		160: //Vision capture tray fiducial 1
			arrStepStatus[7] := 'Step 7: Trigger Vision Capture';
			tonStepTimer(IN:=TRUE, PT:=T#999999S);
			IF NOT G_MachineControl.stMachineOperateMode.DRYRUN THEN
				G_Vision.V20_bRespone := FALSE;
				G_Vision.V20_sSendCmd := 'TRG,2';  
				G_Vision.V20_bTrigger := TRUE;	
			END_IF			
			iStep := 170;
		
		170: //Waiting vision capture done
			tonTimeOut(IN:= TRUE,PT:= tTimeOut);
			IF G_Vision.V20_bRespone OR G_MachineControl.stMachineOperateMode.DRYRUN THEN
				tonTimeOut(IN:= FALSE);
				G_Vision.V20_bTrigger := FALSE;
				arrStepUsedTime[7] := tonStepTimer.ET;
				tonStepTimer(IN:=FALSE);
				iStep := 180;
			ELSIF tonTimeOut.Q THEN
				tonTimeOut(IN:= FALSE);
				G_Vision.V20_bTrigger := FALSE;	
				G_Error.E20_VisionTimeOutInspection	:= TRUE;
				iStep := 160;
			END_IF
			
		180:
			G_Robot.RobotKukaCmd.rRobotPlace_X := G_Values.VA20_stTrayPosition.stFiducialDistance2Value.Xpos;
			G_Robot.RobotKukaCmd.rRobotPlace_Y := G_Values.VA20_stTrayPosition.stFiducialDistance2Value.Ypos;
			G_Robot.RobotKukaCmd.rRobotPlace_Z := 0; //G_Values.VA20_stTrayPosition.stFiducialDistance2Value.Zpos;
			G_Robot.RobotKukaCmd.rRobotPlace_A := G_Values.VA20_stTrayPosition.stFiducialDistance2Value.Apos;
			iStep := 190;
			
		190: //Robot move to tray fiducial 2
			arrStepStatus[8] := 'Step 8: Robot go to tray fiducial 2';
			tonStepTimer(IN:=TRUE, PT:=T#999999S);
			G_Robot.RobotKukaCmd.bRobotTrayFiducial2 := TRUE;
			iStep := 200; 
			
		200:
			IF NOT G_Robot.RobotKukaCmd.bRobotTrayFiducial2Done THEN
				iStep := 210;
			END_IF
			
		210://Robot move tray fiducial 2 done
			tonTimeOut(IN:= TRUE,PT:= tTimeOut);
			IF G_Robot.RobotKukaCmd.bRobotTrayFiducial2Done THEN
				tonTimeOut(IN:= FALSE);
				G_Robot.RobotKukaCmd.bRobotTrayFiducial2 := FALSE;
				arrStepUsedTime[8] := tonStepTimer.ET;
				tonStepTimer(IN:=FALSE);
				iStep := 220;
			ELSIF tonTimeOut.Q THEN
				tonTimeOut(IN:= FALSE);
				G_Robot.RobotKukaCmd.bRobotTrayFiducial2 := FALSE;
				G_Error.E20_RobotTimeOutFailToTrayFiducial_2 := TRUE;
				iStep := 180;
			END_IF
			
		220: //Vision capture tray fiducial 2
			arrStepStatus[9] := 'Step 9: Trigger Vision Capture';
			tonStepTimer(IN:=TRUE, PT:=T#999999S);
			IF NOT G_MachineControl.stMachineOperateMode.DRYRUN THEN
				G_Vision.V20_bRespone := FALSE;
				G_Vision.V20_sSendCmd := 'TRG,3'; 
				G_Vision.V20_bTrigger := TRUE;	
			END_IF				
			iStep := 230;
		
		230: //Waiting vision capture done
			tonTimeOut(IN:= TRUE,PT:= tTimeOut);
			IF G_Vision.V20_bRespone OR G_MachineControl.stMachineOperateMode.DRYRUN THEN
				tonTimeOut(IN:= FALSE);
				G_Vision.V20_bTrigger := FALSE;
				arrStepUsedTime[9] := tonStepTimer.ET;
				tonStepTimer(IN:=FALSE);
				iStep := 240;
			ELSIF tonTimeOut.Q THEN
				tonTimeOut(IN:= FALSE);
				G_Vision.V20_bTrigger := FALSE;	
				G_Error.E20_VisionTimeOutInspection	:= TRUE;
				iStep := 220;
			END_IF
			
		240:
			IF NOT G_MachineControl.stMachineOperateMode.DRYRUN THEN
				G_Robot.RobotKukaCmd.rRobotPlace_X := G_Vision.V20_stTrayPosition.stPocket.Xpos;
				G_Robot.RobotKukaCmd.rRobotPlace_Y := G_Vision.V20_stTrayPosition.stPocket.Ypos;
				G_Robot.RobotKukaCmd.rRobotPlace_Z := G_Values.VA20_rTrayZaxisPick; //G_Vision.V20_stTrayPosition.stPocket.Zpos;
				G_Robot.RobotKukaCmd.rRobotPlace_A := G_Vision.V20_stTrayPosition.stPocket.Apos;
			ELSIF G_MachineControl.stMachineOperateMode.DRYRUN THEN
				G_Robot.RobotKukaCmd.rRobotPlace_X := G_Values.VA20_stTrayPosition.stPocket.Xpos;
				G_Robot.RobotKukaCmd.rRobotPlace_Y := G_Values.VA20_stTrayPosition.stPocket.Ypos;
				G_Robot.RobotKukaCmd.rRobotPlace_Z := G_Values.VA20_rTrayZaxisPick; //G_Values.VA20_stTrayPosition.stPocket.Zpos;
				G_Robot.RobotKukaCmd.rRobotPlace_A := G_Values.VA20_stTrayPosition.stPocket.Apos;
			END_IF
			iStep := 250;
			
		250: //Robot move to pick PCBA
			arrStepStatus[10] := 'Step 10: Robot go to pick PCBA';
			tonStepTimer(IN:=TRUE, PT:=T#999999S);
			G_Robot.RobotKukaCmd.bRobotPickPCBA := TRUE;
			iStep := 260; 
			
		260:
			IF NOT G_Robot.RobotKukaCmd.bRobotPickPCBADone THEN
				iStep := 270;
			END_IF
			
		270://Robot move pick PCBA
			tonTimeOut(IN:= TRUE,PT:= tTimeOut);
			IF G_Robot.RobotKukaCmd.bRobotPickPCBADone THEN
				tonTimeOut(IN:= FALSE);
				G_Auto.A20_bTrayFinish := TRUE;
				G_Robot.RobotKukaCmd.bRobotPickPCBA := FALSE;
				arrStepUsedTime[10] := tonStepTimer.ET;
				tonStepTimer(IN:=FALSE);
				iStep := 280;
			ELSIF tonTimeOut.Q THEN
				tonTimeOut(IN:= FALSE);
				G_Robot.RobotKukaCmd.bRobotPickPCBA := FALSE;
				G_Error.E20_RObotTimeOutFailToPickPCBA := TRUE;
				iStep := 240;
			END_IF
			
		280:
			IF NOT G_MachineControl.stMachineOperateMode.DRYRUN THEN
				G_Robot.RobotKukaCmd.rRobotPlace_X := G_Vision.V20_stPalletPosition.stPocket.Xpos;
				G_Robot.RobotKukaCmd.rRobotPlace_Y := G_Vision.V20_stPalletPosition.stPocket.Ypos;
				G_Robot.RobotKukaCmd.rRobotPlace_Z := G_Values.VA20_rTrayZaxisPick; //G_Vision.V20_stPalletPosition.stPocket.Zpos;
				G_Robot.RobotKukaCmd.rRobotPlace_A := G_Vision.V20_stPalletPosition.stPocket.Apos;
			ELSIF G_MachineControl.stMachineOperateMode.DRYRUN THEN
				G_Robot.RobotKukaCmd.rRobotPlace_X := G_Values.VA20_stPalletPosition.stPocket.Xpos;
				G_Robot.RobotKukaCmd.rRobotPlace_Y := G_Values.VA20_stPalletPosition.stPocket.Ypos;
				G_Robot.RobotKukaCmd.rRobotPlace_Z := G_Values.VA20_rTrayZaxisPick; //G_Values.VA20_stPalletPosition.stPocket.Zpos;
				G_Robot.RobotKukaCmd.rRobotPlace_A := G_Values.VA20_stPalletPosition.stPocket.Apos;
			END_IF
			iStep := 290;
			
		290: //Robot place pcba
			arrStepStatus[11] := 'Step 11: Robot go to place PCBA';
			tonStepTimer(IN:=TRUE, PT:=T#999999S);
			G_Robot.RobotKukaCmd.bRobotPlacePCBA := TRUE;
			iStep := 300;
			
		300:
			IF NOT G_Robot.RobotKukaCmd.bRobotPlacePCBADone THEN
				iStep := 310;
			END_IF
			
		310: //Robot place pcba done
			tonTimeOut(IN:= TRUE,PT:= tTimeOut);
			IF G_Robot.RobotKukaCmd.bRobotPlacePCBADone THEN
				tonTimeOut(IN:= FALSE);
				G_Robot.RobotKukaCmd.bRobotPlacePCBA := FALSE;
				arrStepUsedTime[11] := tonStepTimer.ET;
				tonStepTimer(IN:=FALSE);
				iStep := 320;
			ELSIF tonTimeOut.Q THEN
				tonTimeOut(IN:= FALSE);
				G_Robot.RobotKukaCmd.bRobotPlacePCBA := FALSE;
				G_Error.E20_RobotTimeOutFailToPlacePCBA := TRUE;
				iStep := 280;
			END_IF
			
		320: //Robot go standby pallet
			arrStepStatus[12] := 'Step 12: Robot go to standby';
			tonStepTimer(IN:=TRUE, PT:=T#999999S);
			G_Robot.RobotKukaCmd.bRobotStandbyAtPallet := TRUE;
			iStep := 330;
			
		330:
			IF NOT G_Robot.RobotKukaCmd.bRobotStandbyAtPalletDone THEN
				iStep := 340;
			END_IF
			
		340: //Robot go standby pallet done
			tonTimeOut(IN:= TRUE,PT:= tTimeOut);
			IF G_Robot.RobotKukaCmd.bRobotStandbyAtPalletDone THEN
				tonTimeOut(IN:= FALSE);
				G_Robot.RobotKukaCmd.bRobotStandbyAtPallet := FALSE;
				arrStepUsedTime[12] := tonStepTimer.ET;
				tonStepTimer(IN:=FALSE);
				iStep := 999;
			ELSIF tonTimeOut.Q THEN
				tonTimeOut(IN:= FALSE);
				G_Robot.RobotKukaCmd.bRobotStandbyAtPallet := FALSE;
				G_Error.E20_RobotTimeOutFailToStandbyPallet := TRUE;
				iStep := 280;
			END_IF		
			
		999://Job Done
			G_MachineControl.arrstStationControl[2].bJobDone := TRUE;
			iStep := 0;	
			
		1000: //Robot go to standby at pallet
			//arrStepStatus[7] := 'Step 7: Robot go to place PCBA';
			//tonStepTimer(IN:=TRUE, PT:=T#999999S);
			G_Robot.RobotKukaCmd.bRobotStandbyAtPallet := TRUE;
			iStep := 1010;
			
		1010:
			IF NOT G_Robot.RobotKukaCmd.bRobotStandbyAtPalletDone THEN
				iStep := 1020;
			END_IF
			
		1020: //Robot go to standby pallet done
			tonTimeOut(IN:= TRUE,PT:= tTimeOut);
			IF G_Robot.RobotKukaCmd.bRobotStandbyAtPalletDone THEN
				G_Robot.RobotKukaCmd.bRobotStandbyAtPallet := FALSE;
				G_Auto.A20_bRobotAtStandbyPallet := TRUE;
				iStep := 0;
			ELSIF tonTimeOut.Q THEN
				tonTimeOut(IN:= FALSE);
				G_Robot.RobotKukaCmd.bRobotStandbyAtPallet := FALSE;
				G_Error.E20_RobotTimeOutFailToStandbyPallet := TRUE;
				iStep := 2000;
			END_IF
			
		2000: //Robot go to standby at tray
			//arrStepStatus[7] := 'Step 7: Robot go to place PCBA';
			//tonStepTimer(IN:=TRUE, PT:=T#999999S);
			G_Robot.RobotKukaCmd.bRobotStandbyAtTray := TRUE;
			iStep := 2010;
			
		2010:
			IF NOT G_Robot.RobotKukaCmd.bRobotStandbyAtTrayDone THEN
				iStep := 2020;
			END_IF
			
		2020: //Robot go to standby tray done
			tonTimeOut(IN:= TRUE,PT:= tTimeOut);
			IF G_Robot.RobotKukaCmd.bRobotStandbyAtTrayDone THEN
				G_Robot.RobotKukaCmd.bRobotStandbyAtTray := FALSE;
				G_Auto.A20_bRobotAtStandbyTray := TRUE;
				iStep := 110;
			ELSIF tonTimeOut.Q THEN
				tonTimeOut(IN:= FALSE);
				G_Robot.RobotKukaCmd.bRobotStandbyAtTray := FALSE;
				G_Error.E20_RobotTimeOutFailToStandbyTray := TRUE;
				iStep := 2000;
			END_IF
			
		3000: //Recovery For Failed Overpress
			G_Robot.RobotKukaStandard.bStop := TRUE;	
			tonDelay(IN:=TRUE, PT:=T#2S);
			IF tonDelay.Q THEN
				tonDelay(IN:=FALSE);
				iStep := 3010;
			END_IF
			
		3010:
			G_Robot.RobotKukaStandard.bStop	:= FALSE;
			tonDelay(IN:=TRUE, PT:=T#2S);
			IF tonDelay.Q THEN
				tonDelay(IN:=FALSE);
				iStep := 3020;
			END_IF
			
		3020: //Robot start
			G_Robot.RobotKukaStandard.bStart := TRUE;
			iStep := 3030;
			
		3030: //Wait start
			tonTimeOut(IN:= TRUE, PT:= T#50S);
			IF G_Robot.RobotKukaStandard.bRunning THEN
				tonTimeOut(IN:=FALSE);
				iStep := 3040;
			ELSIF tonTimeOut.Q THEN
				tonTimeOut(IN:=FALSE);
				G_Robot.RobotKukaStandard.bStart := FALSE;
				G_Error.E20_RobotFailStart := TRUE;	
				iStep := 3020;
			END_IF
			
		3040: //Robot StandbyPosition
			G_Robot.RobotKukaStandard.bHome := TRUE;
			iStep := 3050;
			
		3050:
			IF NOT G_Robot.RobotKukaStandard.bHomeDone THEN
				iStep := 3060;
			END_IF
 
		3060: //Wait home
			tonTimeOut(IN:= TRUE, PT:= T#500S);
			IF G_Robot.RobotKukaStandard.bHomeDone THEN
				G_Robot.RobotKukaStandard.bHome := FALSE;
				G_Error.E20_RobotFailPlaceOverpress := TRUE;
				tonTimeOut(IN:=FALSE);
				iStep := 999;	
			ELSIF tonTimeOut.Q THEN
				tonTimeOut(IN:=FALSE);
				G_Robot.RobotKukaStandard.bHome := FALSE;
				G_Error.E20_RobotFailHome := TRUE;
				iStep := 3040;
			END_IF
			
	END_CASE

END_IF

FOR iMatching := 1 TO 100 DO
	G_MachineControl.arrsST20StepStatus[iMatching] := arrStepStatus[iMatching];
	G_MachineControl.arrtimeST20StepTime[iMatching] := arrStepUsedTime[iMatching];
END_FOR

END_PROGRAM

// ---- POUs/General/DoorLock.TcPOU
PROGRAM DoorLock
VAR
END_VAR

END_PROGRAM

// ---- POUs/General/NewLotEndLot.TcPOU
PROGRAM NewLotEndLot
VAR
	bLotStart: BOOL;
	RTRIG_EndLot : R_TRIG;
	iStepEndLot : INT;
END_VAR

//=================================
//New Lot Confirm
//=================================
IF (G_Manual.M_bNewLotConfirm AND NOT bLotStart) OR G_Manual.M_bLoadRecipe THEN
	G_Values.VA20_byteRobotProgramID := G_Recipe.R20_byteRobotProgramID;
	G_Values.VA20_stTrayPosition := G_Recipe.R20_stTrayPosition;
	G_Values.VA20_stPalletPosition := G_Recipe.R20_stPalletPosition;
	G_Values.VA20_rTrayZaxisPick := G_Recipe.R20_rTrayZaxisPick;
	G_Values.VA20_rPalletZaxisPlace := G_Recipe.R20_rPalletZaxisPlace;
//	G_Values.VA00_rConveyorWidth := G_Recipe.R00_rConveyorWidth; //to do
	G_Auto.A20_bRobotChangeRecipe := TRUE;
	G_Manual.M_bLoadRecipe := FALSE;
	IF G_Manual.M_bNewLotConfirm THEN
		bLotStart := TRUE;
	END_IF
END_IF

IF bLotStart AND G_Auto.A20_bRobotChangeRecipeDone THEN
	G_Manual.M_bLotStarted := TRUE;
	G_Manual.M_bNewLotConfirm := FALSE;
	G_Manual.M_bEndLot := FALSE;
	bLotStart := FALSE;
END_IF


RTRIG_EndLot(CLK:= G_Manual.M_bEndLot);

IF RTRIG_EndLot.Q THEN
	iStepEndLot := 10;
END_IF

CASE iStepEndLot OF
	
10:
	IF G_MachineControl.arrstStationControl[2].bJobDone AND G_MachineControl.arrstStationControl[3].bJobDone AND G_MachineControl.arrstStationControl[4].bJobDone THEN
		;// to do conveyor handle
		iStepEndLot := 20;
	END_IF

20:
	G_Home.H20_bHome := TRUE;
	iStepEndLot := 30;
	
30:
	IF G_Home.H20_bHomeDone THEN
		iStepEndLot := 40;
	END_IF
	
40:
	G_Manual.M_bStart := FALSE;
	G_Manual.M_bStop := TRUE;
	iStepEndLot := 50;
	
50:
	G_Manual.M_bEndLot := FALSE;
	G_Manual.M_bLotStarted := FALSE;
	bLotStart := FALSE;
	iStepEndLot := 0;
END_CASE

END_PROGRAM

// ---- POUs/Station/ST20_PickNPlace/Robot/ST20_VisionManualControl.TcPOU
PROGRAM ST20_VisionManualControl
VAR
END_VAR

IF G_MachineControl.stMachineOperateMode.MANUAL THEN
	
	IF G_Manual.M20_bVisionTrayFiducial1 THEN
		G_Vision.V20_bRespone := FALSE;
		G_Vision.V20_sSendCmd := 'TRG,0';
		G_Vision.V20_bTrigger := TRUE;
		G_Manual.M20_bVisionTrayFiducial1 := FALSE;	
	END_IF
	
	IF G_Manual.M20_bVisionTrayFiducial2 THEN
		G_Vision.V20_bRespone := FALSE;
		G_Vision.V20_sSendCmd := 'TRG,1';
		G_Vision.V20_bTrigger := TRUE;
		G_Manual.M20_bVisionTrayFiducial2 := FALSE;	
	END_IF
	
	IF G_Manual.M20_bVisionPalletFiducial1 THEN
		G_Vision.V20_bRespone := FALSE;
		G_Vision.V20_sSendCmd := 'TRG,2';
		G_Vision.V20_bTrigger := TRUE;
		G_Manual.M20_bVisionPalletFiducial1 := FALSE;	
	END_IF
	
	IF G_Manual.M20_bVisionPalletFiducial2 THEN
		G_Vision.V20_bRespone := FALSE;
		G_Vision.V20_sSendCmd := 'TRG,3';
		G_Vision.V20_bTrigger := TRUE;
		G_Manual.M20_bVisionPalletFiducial2 := FALSE;	
	END_IF
	
END_IF

END_PROGRAM
